(* Logix 5000 project; controller NSutherlandCapstone Emulate 5570 rev 32.11; software revision 32.00; part 2 of 2 *)
(* tags used below, declared in another part *)
   A : BOOL;
   AndOr_SetBit : SFC_STEP;
   AndOr_SetDone : BOOL;
   AndOr_SetPL1 : SFC_ACTION;
   AndOr_SetPL2 : SFC_ACTION;
   AndOr_SetPL3 : SFC_ACTION;
   AndOr_SetPL4 : SFC_ACTION;
   B : BOOL;
   C : BOOL;
   CARRY_OUT : BOOL;
   FullAdder_SetBit : SFC_STEP;
   FullAdder_SetCarry : SFC_ACTION;
   FullAdder_SetDone : BOOL;
   FullAdder_SetSum : SFC_ACTION;
   OutputNOR : BOOL;
   OutputXOR : BOOL;
   PB1 : BOOL;   // NO PB
   PB2 : BOOL;   // NC PB
   PB3 : BOOL;   // NC PB
   PB4 : BOOL;   // NO PB
   PL1 : BOOL;
   PL2 : BOOL;
   PL3 : BOOL;
   PL4 : BOOL;
   SUM_OUT : BOOL;
   TruthTables_SetBit : SFC_STEP;
   TruthTables_SetDone : BOOL;
   TruthTables_SetNOR : SFC_ACTION;
   TruthTables_SetXOR : SFC_ACTION;
   XICXIO_SetBit : SFC_STEP;
   XICXIO_SetDone : BOOL;
   XICXIO_SetPL1 : SFC_ACTION;
   XICXIO_SetPL2 : SFC_ACTION;
   XICXIO_SetPL3 : SFC_ACTION;
   XICXIO_SetPL4 : SFC_ACTION;
   SS : BOOL;
(* MainProgram, continued *)

ROUTINE FBD_2_AndOr   (* function block diagram *)
   SHEET 1
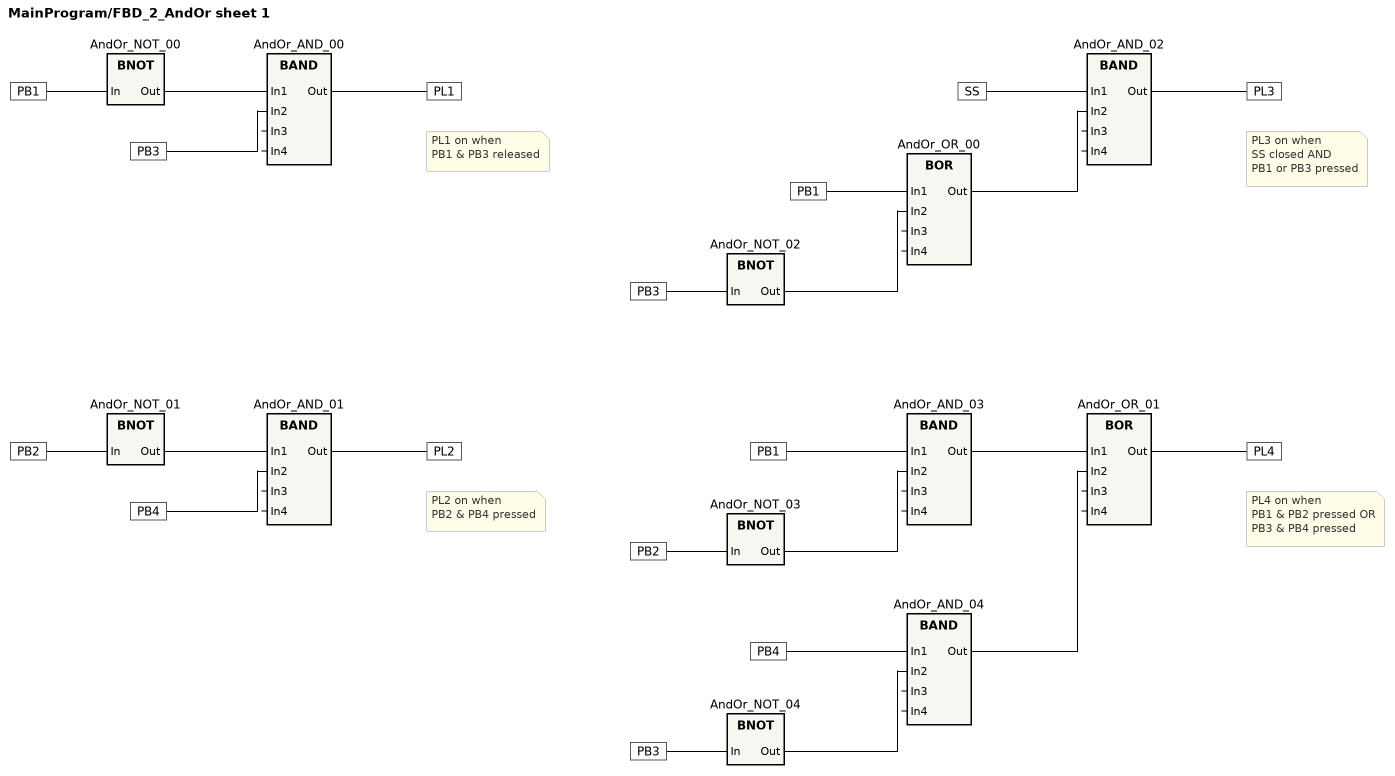
   AndOr_NOT_00 : BNOT(In := PB1);
   AndOr_NOT_01 : BNOT(In := PB2);
   AndOr_AND_00 : BAND(In1 := AndOr_NOT_00.Out, In2 := PB3);   // unwired pins: In3 In4
   AndOr_AND_01 : BAND(In1 := AndOr_NOT_01.Out, In2 := PB4);   // unwired pins: In3 In4
   // PL1 on when
   // PB1 & PB3 released
   PL1 := AndOr_AND_00.Out;
   // PL2 on when
   // PB2 & PB4 pressed
   PL2 := AndOr_AND_01.Out;
   AndOr_NOT_02 : BNOT(In := PB3);
   AndOr_NOT_03 : BNOT(In := PB2);
   AndOr_NOT_04 : BNOT(In := PB3);
   AndOr_OR_00 : BOR(In1 := PB1, In2 := AndOr_NOT_02.Out);   // unwired pins: In3 In4
   AndOr_AND_03 : BAND(In1 := PB1, In2 := AndOr_NOT_03.Out);   // unwired pins: In3 In4
   AndOr_AND_04 : BAND(In1 := PB4, In2 := AndOr_NOT_04.Out);   // unwired pins: In3 In4
   AndOr_AND_02 : BAND(In1 := SS, In2 := AndOr_OR_00.Out);   // unwired pins: In3 In4
   AndOr_OR_01 : BOR(In1 := AndOr_AND_03.Out, In2 := AndOr_AND_04.Out);   // unwired pins: In3 In4
   // PL3 on when
   // SS closed AND
   // PB1 or PB3 pressed
   PL3 := AndOr_AND_02.Out;
   // PL4 on when
   // PB1 & PB2 pressed OR
   // PB3 & PB4 pressed
   PL4 := AndOr_OR_01.Out;
END_ROUTINE

ROUTINE FBD_3_TruthTables   (* function block diagram *)
   SHEET 1
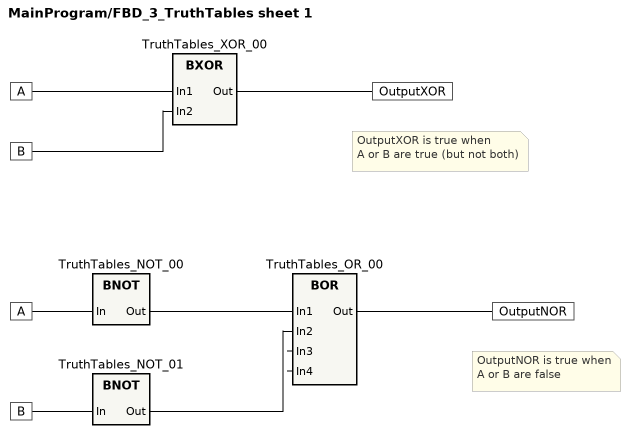
   TruthTables_NOT_00 : BNOT(In := A);
   TruthTables_NOT_01 : BNOT(In := B);
   TruthTables_XOR_00 : BXOR(In1 := A, In2 := B);
   TruthTables_OR_00 : BOR(In1 := TruthTables_NOT_00.Out, In2 := TruthTables_NOT_01.Out);   // unwired pins: In3 In4
   // OutputXOR is true when
   // A or B are true (but not both)
   OutputXOR := TruthTables_XOR_00.Out;
   // OutputNOR is true when
   // A or B are false
   OutputNOR := TruthTables_OR_00.Out;
END_ROUTINE

ROUTINE FBD_4_FullAdder   (* function block diagram *)
   SHEET 1
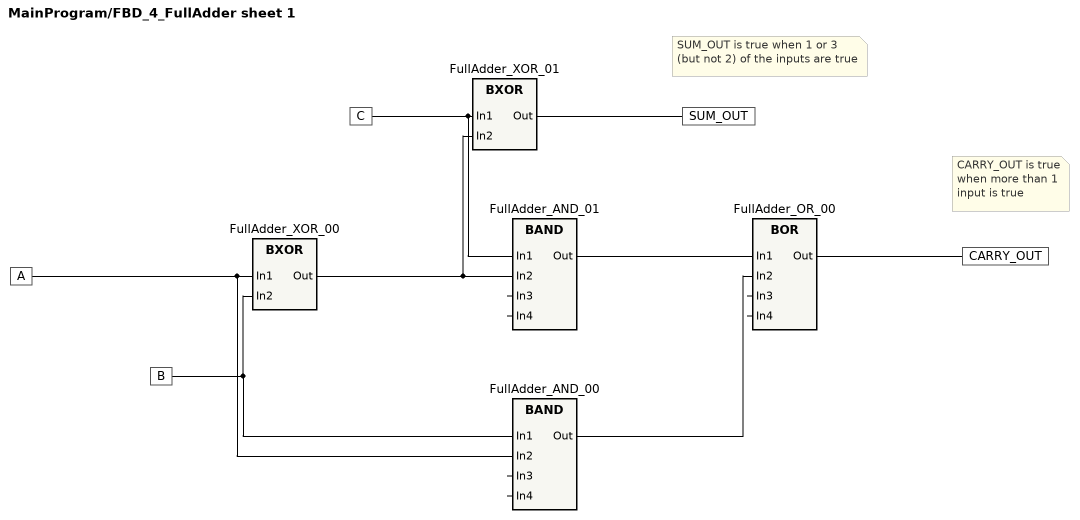
   FullAdder_XOR_00 : BXOR(In1 := A, In2 := B);
   FullAdder_XOR_01 : BXOR(In1 := C, In2 := FullAdder_XOR_00.Out);
   FullAdder_AND_01 : BAND(In1 := C, In2 := FullAdder_XOR_00.Out);   // unwired pins: In3 In4
   FullAdder_AND_00 : BAND(In1 := B, In2 := A);   // unwired pins: In3 In4
   // SUM_OUT is true when 1 or 3
   // (but not 2) of the inputs are true
   SUM_OUT := FullAdder_XOR_01.Out;
   FullAdder_OR_00 : BOR(In1 := FullAdder_AND_01.Out, In2 := FullAdder_AND_00.Out);   // unwired pins: In3 In4
   // CARRY_OUT is true
   // when more than 1
   // input is true
   CARRY_OUT := FullAdder_OR_00.Out;
END_ROUTINE

ROUTINE MainRoutine   (* structured text *)
   JSR(ST_2_AndOr); // Calls desired subroutine
END_ROUTINE

ROUTINE SFC_1_XICXIO   (* sequential function chart *)
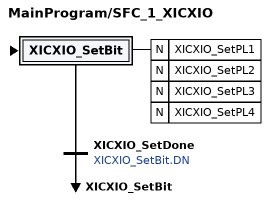
   INITIAL_STEP XICXIO_SetBit:
      ACTION XICXIO_SetPL1 (N):
         PL1 := PB1;
      END_ACTION
      ACTION XICXIO_SetPL2 (N):
         PL2 := NOT PB2;
      END_ACTION
      ACTION XICXIO_SetPL3 (N):
         PL3 := PB3;
      END_ACTION
      ACTION XICXIO_SetPL4 (N):
         PL4 := NOT PB4;
      END_ACTION
   END_STEP
   TRANSITION XICXIO_SetDone FROM XICXIO_SetBit TO XICXIO_SetBit
      := XICXIO_SetBit.DN
   END_TRANSITION
END_ROUTINE

ROUTINE SFC_2_AndOr   (* sequential function chart *)
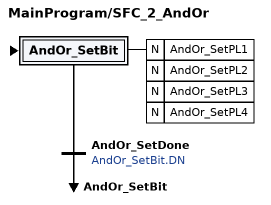
   INITIAL_STEP AndOr_SetBit:
      ACTION AndOr_SetPL1 (N):
         PL1 := NOT PB1 & PB3;
      END_ACTION
      ACTION AndOr_SetPL2 (N):
         PL2 := NOT PB2 OR PB4;
      END_ACTION
      ACTION AndOr_SetPL3 (N):
         PL3 := SS & (PB1 OR NOT PB3);
      END_ACTION
      ACTION AndOr_SetPL4 (N):
         PL4 := (PB1 & NOT PB2) OR
         	   (NOT PB3 & PB4);
      END_ACTION
   END_STEP
   TRANSITION AndOr_SetDone FROM AndOr_SetBit TO AndOr_SetBit
      := AndOr_SetBit.DN
   END_TRANSITION
END_ROUTINE

ROUTINE SFC_3_TruthTables   (* sequential function chart *)
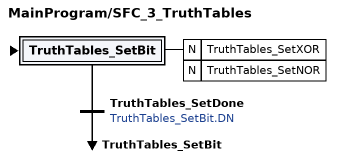
   INITIAL_STEP TruthTables_SetBit:
      ACTION TruthTables_SetXOR (N):
         OutputXOR := A XOR B;
      END_ACTION
      ACTION TruthTables_SetNOR (N):
         OutputNOR := NOT A OR NOT B;
      END_ACTION
   END_STEP
   TRANSITION TruthTables_SetDone FROM TruthTables_SetBit TO TruthTables_SetBit
      := TruthTables_SetBit.DN
   END_TRANSITION
END_ROUTINE

ROUTINE SFC_4_FullAdder   (* sequential function chart *)
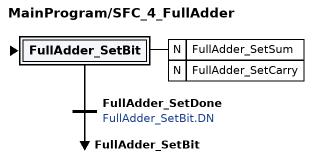
   INITIAL_STEP FullAdder_SetBit:
      ACTION FullAdder_SetSum (N):
         SUM_OUT := (NOT A & NOT B & C) OR
         		   (NOT A & B & NOT C) OR
         		   (A & NOT B & NOT C) OR
         		   (A & B & C);
      END_ACTION
      ACTION FullAdder_SetCarry (N):
         CARRY_OUT := (NOT A & B & C) OR
         			 (A & NOT B & C) OR
         			 (A & B & NOT C) OR
         			 (A & B & C);
      END_ACTION
   END_STEP
   TRANSITION FullAdder_SetDone FROM FullAdder_SetBit TO FullAdder_SetBit
      := FullAdder_SetBit.DN
   END_TRANSITION
END_ROUTINE

ROUTINE ST_1_XICXIO   (* structured text *)
// Routine 1 of PLC Lab 2
   // Lab 2 R1_XICXIO
   (*	PB1 = NO
   	PB2 = NC
   	PB3 = NC
   	PB4 = NO *)
   
   PL1 := PB1;			// PL1 on when PB1 pressed
   PL2 := NOT PB2;		// PL2 on when PB2 pressed
   PL3 := PB3;			// PL3 off when PB3 pressed
   PL4 := NOT PB4;		// PL4 off when PB4 pressed
END_ROUTINE

ROUTINE ST_2_AndOr   (* structured text *)
// Routine 2 of PLC Lab 2
   // Lab 2 R2_AndOr
   (*	PB1 = NO
   	PB2 = NC
   	PB3 = NC
   	PB4 = NO *)
   
   PL1 := NOT PB1 & PB3;			// PL1 on when PB1 & PB3 released
   PL2 := NOT PB2 OR PB4;			// PL2 on when PB2 or PB4 pressed
   PL3 := SS & (PB1 OR NOT PB3);	// PL3 on when SS closed & PB1 or PB3 pressed
   PL4 := (PB1 & NOT PB2) OR		// PL4 on when PB1 & PB2 pressed or PB3 & PB4 pressed
   	   (NOT PB3 & PB4);
END_ROUTINE

ROUTINE ST_3_TruthTables   (* structured text *)
// Routine 3 of PLC Lab 2
   // Lab 2 R3_TruthTable
   
   OutputXOR := A XOR B;		// True when A or B are 1 (but not both)
   OutputNOR := NOT A OR NOT B;	// True when A and/or B are 0
END_ROUTINE

ROUTINE ST_4_FullAdder   (* structured text *)
// Routine 4 of PLC Lab 2 (BONUS)
   // LAB 2 R4_FullAdder
   (*
   	A	B	C		SUM_OUT	CARRY_OUT
   	0	0	1			1		0
   	0	1	0			1		0
   	1	0	0			1		0
   	1	1	1			1		1
   	0	1	1			0		1
   	1	1	0			0		1
   	1	0	1			0		1
   *)
   
   SUM_OUT   := (NOT A & NOT B & C) OR
   			 (NOT A & B & NOT C) OR
   			 (A & NOT B & NOT C) OR
   			 (A & B & C);
   
   CARRY_OUT := (NOT A & B & C) OR
   			 (A & NOT B & C) OR
   			 (A & B & NOT C) OR
   			 (A & B & C);
END_ROUTINE
END_PROGRAM
